TYPE LAxisCtrl_typeJog :
STRUCT
	velocity			:LREAL;
	acceleration		:LREAL;
	deceleration		:LREAL;
	jerk				:LREAL;
	positionControlled	:BOOL;
	increment			:LREAL;
	mode				:DINT;

END_STRUCT
END_TYPE

(* stored: Version 1.1.0.1
   DUT LAxisCtrl_typeJog: Id {85b02d6b-8baf-4572-a4df-5c7c27c01b85} *)
